// TIA Portal project "PLC - Mo hinh chiet rot" (V15)

(* hardware
DEVICE "S7-1200 station_1"  S7-1200 Station
   slot 0: "Rack_0"  S7-1200 Rack  Rack  V1.0
   slot 1: "PLC_1"  CPU 1212C AC/DC/Rly  6ES7 212-1BE40-0XB0  V4.2
   slot 2: "DQ 8xRelay_1"  SM 1222 DQ8 x relay  6ES7 222-1HF32-0XB0  V2.0
*)

// ===== PLC "PLC_1"  CPU 1212C AC/DC/Rly =====

VAR_GLOBAL   // PLC tag table "Default tag table"
   "CB1" AT %I0.0 : Bool;
   "CB2" AT %I0.1 : Bool;
   "CB3" AT %I0.2 : Bool;
   "CB4" AT %I0.3 : Bool;
   "Start" AT %I0.4 : Bool;
   "Stop" AT %I0.5 : Bool;
   "Reset" AT %I0.6 : Bool;
   "Emc" AT %I0.7 : Bool;
   "Van1" AT %Q0.0 : Bool;
   "Van2" AT %Q0.1 : Bool;
   "Van3" AT %Q0.2 : Bool;
   "Van4" AT %Q0.3 : Bool;
   "Van5" AT %Q0.4 : Bool;
   "Van6" AT %Q0.5 : Bool;
   "Step-M-MXoay" AT %Q1.0 : Bool;
   "Step-U-Dnhan" AT %Q1.7 : Bool;
   "DC1-M-BT1" AT %Q1.3 : Bool;
   "DC2-M-BT2" AT %Q1.4 : Bool;
   "DC3-M-CNap" AT %Q1.5 : Bool;
   "DC4-M-Bom" AT %Q1.6 : Bool;
   "DC5-U-BT3" AT %Q1.1 : Bool;
   "M-Start" AT %M0.0 : Bool;
   "M-Start3s" AT %M1.0 : Bool;
   "M-Bom" AT %M2.0 : Bool;
   "M-MX chay dien" AT %M1.1 : Bool;
   "M-MX chay" AT %M2.1 : Bool;
   "Tag_1" AT %M4.1 : Bool;
   "Tag_3" AT %M4.2 : Bool;
   "Tag_4" AT %MW10 : Int;
   "Tag_5" AT %M4.5 : Bool;
   "Tag_6" AT %M0.1 : Bool;
   "Tag_7" AT %M0.2 : Bool;
   "Tag_8" AT %M0.3 : Bool;
   "Tag_9" AT %M0.5 : Bool;
   "Tag_2" AT %M6.0 : Bool;
   "Tag_10" AT %M0.4 : Bool;
   "Tag_11" AT %M9.0 : Bool;
END_VAR

// folder: System blocks/Program resources

DATA_BLOCK "t1"   // DB1
{ S7_Optimized_Access := 'TRUE' }
AUTHOR : Simatic
FAMILY : IEC
NAME : IEC_TMR
VERSION : 1.0
// stored: InstanceOfName IEC_TIMER
"IEC_TIMER"
BEGIN
END_DATA_BLOCK

DATA_BLOCK "t2"   // DB2
{ S7_Optimized_Access := 'TRUE' }
AUTHOR : Simatic
FAMILY : IEC
NAME : IEC_TMR
VERSION : 1.0
// stored: InstanceOfName IEC_TIMER
"IEC_TIMER"
BEGIN
END_DATA_BLOCK

DATA_BLOCK "T0"   // DB3
{ S7_Optimized_Access := 'TRUE' }
AUTHOR : Simatic
FAMILY : IEC
NAME : IEC_TMR
VERSION : 1.0
// stored: InstanceOfName IEC_TIMER
"IEC_TIMER"
BEGIN
END_DATA_BLOCK

DATA_BLOCK "t3"   // DB4
{ S7_Optimized_Access := 'TRUE' }
AUTHOR : Simatic
FAMILY : IEC
NAME : IEC_TMR
VERSION : 1.0
// stored: InstanceOfName IEC_TIMER
"IEC_TIMER"
BEGIN
END_DATA_BLOCK

DATA_BLOCK "t9"   // DB5
{ S7_Optimized_Access := 'TRUE' }
AUTHOR : Simatic
FAMILY : IEC
NAME : IEC_TMR
VERSION : 1.0
// stored: InstanceOfName IEC_TIMER
"IEC_TIMER"
BEGIN
END_DATA_BLOCK

DATA_BLOCK "t5"   // DB6
{ S7_Optimized_Access := 'TRUE' }
AUTHOR : Simatic
FAMILY : IEC
NAME : IEC_TMR
VERSION : 1.0
// stored: InstanceOfName IEC_TIMER
"IEC_TIMER"
BEGIN
END_DATA_BLOCK

DATA_BLOCK "t6"   // DB7
{ S7_Optimized_Access := 'TRUE' }
AUTHOR : Simatic
FAMILY : IEC
NAME : IEC_TMR
VERSION : 1.0
// stored: InstanceOfName IEC_TIMER
"IEC_TIMER"
BEGIN
END_DATA_BLOCK

DATA_BLOCK "t7"   // DB8
{ S7_Optimized_Access := 'TRUE' }
AUTHOR : Simatic
FAMILY : IEC
NAME : IEC_TMR
VERSION : 1.0
// stored: InstanceOfName IEC_TIMER
"IEC_TIMER"
BEGIN
END_DATA_BLOCK

DATA_BLOCK "t8"   // DB9
{ S7_Optimized_Access := 'TRUE' }
AUTHOR : Simatic
FAMILY : IEC
NAME : IEC_TMR
VERSION : 1.0
// stored: InstanceOfName IEC_TIMER
"IEC_TIMER"
BEGIN
END_DATA_BLOCK

DATA_BLOCK "t10"   // DB10
{ S7_Optimized_Access := 'TRUE' }
AUTHOR : Simatic
FAMILY : IEC
NAME : IEC_TMR
VERSION : 1.0
// stored: InstanceOfName IEC_TIMER
"IEC_TIMER"
BEGIN
END_DATA_BLOCK

DATA_BLOCK "dem"   // DB11
{ S7_Optimized_Access := 'TRUE' }
AUTHOR : Simatic
FAMILY : IEC
NAME : CNTR
VERSION : 1.0
// stored: InstanceOfName IEC_COUNTER
"IEC_COUNTER"
BEGIN
END_DATA_BLOCK

DATA_BLOCK "t11"   // DB12
{ S7_Optimized_Access := 'TRUE' }
AUTHOR : Simatic
FAMILY : IEC
NAME : IEC_TMR
VERSION : 1.0
// stored: InstanceOfName IEC_TIMER
"IEC_TIMER"
BEGIN
END_DATA_BLOCK

DATA_BLOCK "t24"   // DB13
{ S7_Optimized_Access := 'TRUE' }
AUTHOR : Simatic
FAMILY : IEC
NAME : IEC_TMR
VERSION : 1.0
// stored: InstanceOfName IEC_TIMER
"IEC_TIMER"
BEGIN
END_DATA_BLOCK

DATA_BLOCK "t12"   // DB14
{ S7_Optimized_Access := 'TRUE' }
AUTHOR : Simatic
FAMILY : IEC
NAME : IEC_TMR
VERSION : 1.0
// stored: InstanceOfName IEC_TIMER
"IEC_TIMER"
BEGIN
END_DATA_BLOCK

DATA_BLOCK "t25"   // DB15
{ S7_Optimized_Access := 'TRUE' }
AUTHOR : Simatic
FAMILY : IEC
NAME : IEC_TMR
VERSION : 1.0
// stored: InstanceOfName IEC_TIMER
"IEC_TIMER"
BEGIN
END_DATA_BLOCK

DATA_BLOCK "t13"   // DB16
{ S7_Optimized_Access := 'TRUE' }
AUTHOR : Simatic
FAMILY : IEC
NAME : IEC_TMR
VERSION : 1.0
// stored: InstanceOfName IEC_TIMER
"IEC_TIMER"
BEGIN
END_DATA_BLOCK

DATA_BLOCK "t16"   // DB17
{ S7_Optimized_Access := 'TRUE' }
AUTHOR : Simatic
FAMILY : IEC
NAME : IEC_TMR
VERSION : 1.0
// stored: InstanceOfName IEC_TIMER
"IEC_TIMER"
BEGIN
END_DATA_BLOCK

DATA_BLOCK "t23"   // DB18
{ S7_Optimized_Access := 'TRUE' }
AUTHOR : Simatic
FAMILY : IEC
NAME : IEC_TMR
VERSION : 1.0
// stored: InstanceOfName IEC_TIMER
"IEC_TIMER"
BEGIN
END_DATA_BLOCK

DATA_BLOCK "t20"   // DB19
{ S7_Optimized_Access := 'TRUE' }
AUTHOR : Simatic
FAMILY : IEC
NAME : IEC_TMR
VERSION : 1.0
// stored: InstanceOfName IEC_TIMER
"IEC_TIMER"
BEGIN
END_DATA_BLOCK

DATA_BLOCK "t26"   // DB20
{ S7_Optimized_Access := 'TRUE' }
AUTHOR : Simatic
FAMILY : IEC
NAME : IEC_TMR
VERSION : 1.0
// stored: InstanceOfName IEC_TIMER
"IEC_TIMER"
BEGIN
END_DATA_BLOCK

DATA_BLOCK "t27"   // DB21
{ S7_Optimized_Access := 'TRUE' }
AUTHOR : Simatic
FAMILY : IEC
NAME : IEC_TMR
VERSION : 1.0
// stored: InstanceOfName IEC_TIMER
"IEC_TIMER"
BEGIN
END_DATA_BLOCK

// folder: (top level)

ORGANIZATION_BLOCK "Main"   // OB1, LAD, ProgramCycle
TITLE = "Main Program Sweep (Cycle)"
{ S7_Optimized_Access := 'TRUE' }
VERSION : 0.1
   VAR_INPUT
      Initial_Call : Bool;   // Initial call of this OB
      Remanence : Bool;   // =True, if remanent data are available
   END_VAR
   VAR_TEMP   // added for the SCL form of the ladder/FBD networks
      _w1 : Bool;
   END_VAR
BEGIN

REGION Network 1: start vs stop
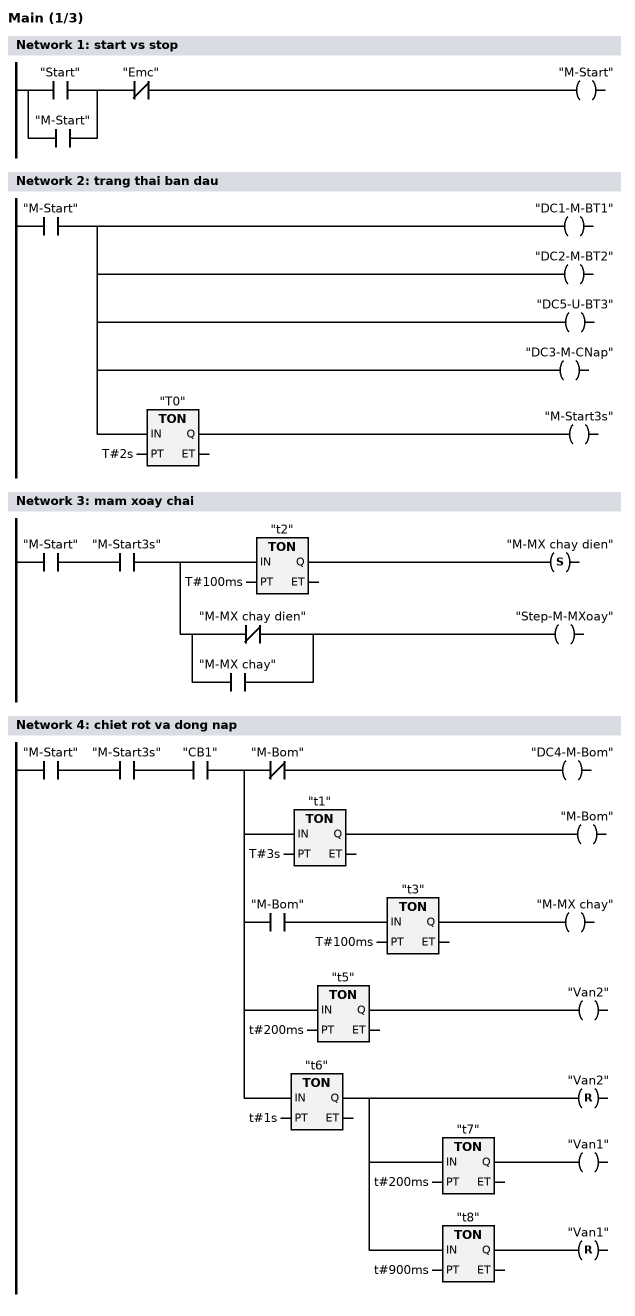
   RUNG wire#powerrail
      Contact( "Start" )
      wire#w1
      I_Contact( "Emc" )
      Coil( "M-Start" )
   END_RUNG
   RUNG wire#powerrail
      Contact( "M-Start" )
   END_RUNG wire#w1
   // the same network as SCL:
   "M-Start" := ("Start" OR "M-Start") AND NOT "Emc";
END_REGION

REGION Network 2: trang thai ban dau
   "DC1-M-BT1" := "M-Start";
   "DC2-M-BT2" := "M-Start";
   "DC5-U-BT3" := "M-Start";
   "DC3-M-CNap" := "M-Start";
   "T0".TON(IN := "M-Start", PT := T#2s);
   "M-Start3s" := "T0".Q;
END_REGION

REGION Network 3: mam xoay chai
   #_w1 := "M-Start" AND "M-Start3s";
   "t2".TON(IN := #_w1, PT := T#100ms);
   IF "t2".Q THEN "M-MX chay dien" := TRUE; END_IF;
   "Step-M-MXoay" := #_w1 AND (NOT "M-MX chay dien" OR "M-MX chay");
END_REGION

REGION Network 4: chiet rot va dong nap
   #_w1 := "M-Start" AND "M-Start3s" AND "CB1";
   "DC4-M-Bom" := #_w1 AND NOT "M-Bom";
   "t1".TON(IN := #_w1, PT := T#3s);
   "M-Bom" := "t1".Q;
   "t3".TON(IN := #_w1 AND "M-Bom", PT := T#100ms);
   "M-MX chay" := "t3".Q;
   "t5".TON(IN := #_w1, PT := t#200ms);
   "Van2" := "t5".Q;
   "t6".TON(IN := #_w1, PT := t#1s);
   IF "t6".Q THEN "Van2" := FALSE; END_IF;
   "t7".TON(IN := "t6".Q, PT := t#200ms);
   "Van1" := "t7".Q;
   "t8".TON(IN := "t6".Q, PT := t#900ms);
   IF "t8".Q THEN "Van1" := FALSE; END_IF;
END_REGION

REGION Network 5
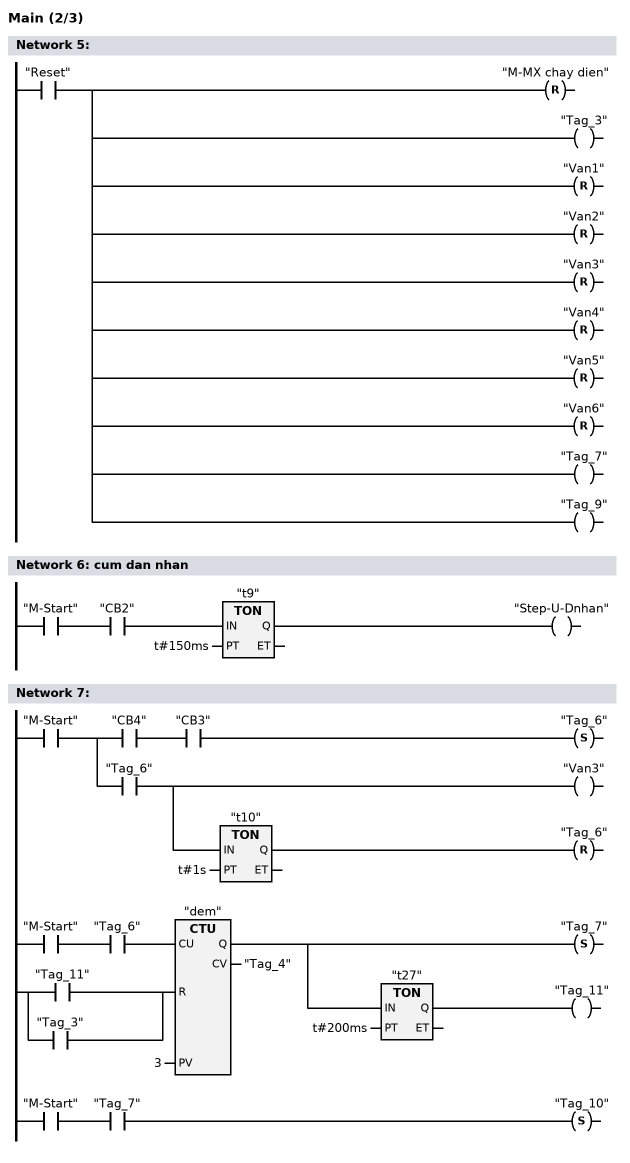
   RUNG wire#powerrail
      Contact( "Reset" )
      wire#w1
      R_Coil( "M-MX chay dien" )
   END_RUNG
   RUNG wire#w1
      Coil( "Tag_3" )
   END_RUNG
   RUNG wire#w1
      R_Coil( "Van1" )
   END_RUNG
   RUNG wire#w1
      R_Coil( "Van2" )
   END_RUNG
   RUNG wire#w1
      R_Coil( "Van3" )
   END_RUNG
   RUNG wire#w1
      R_Coil( "Van4" )
   END_RUNG
   RUNG wire#w1
      R_Coil( "Van5" )
   END_RUNG
   RUNG wire#w1
      R_Coil( "Van6" )
   END_RUNG
   RUNG wire#w1
      Coil( "Tag_7" )
   END_RUNG
   RUNG wire#w1
      Coil( "Tag_9" )
   END_RUNG
   // the same network as SCL:
   IF "Reset" THEN "M-MX chay dien" := FALSE; END_IF;
   "Tag_3" := "Reset";
   IF "Reset" THEN
       "Van1" := FALSE;
       "Van2" := FALSE;
       "Van3" := FALSE;
       "Van4" := FALSE;
       "Van5" := FALSE;
       "Van6" := FALSE;
   END_IF;
   "Tag_7" := "Reset";
   "Tag_9" := "Reset";
END_REGION

REGION Network 6: cum dan nhan
   "t9".TON(IN := "M-Start" AND "CB2", PT := t#150ms);
   "Step-U-Dnhan" := "t9".Q;
END_REGION

REGION Network 7
   IF "M-Start" AND "CB4" AND "CB3" THEN "Tag_6" := TRUE; END_IF;
   "Van3" := "M-Start" AND "Tag_6";
   "t10".TON(IN := "Van3", PT := t#1s);
   IF "t10".Q THEN "Tag_6" := FALSE; END_IF;
   "dem".CTU(CU := "M-Start" AND "Tag_6", R := "Tag_11" OR "Tag_3", PV := 3, CV => "Tag_4");
   IF "dem".Q THEN "Tag_7" := TRUE; END_IF;
   "t27".TON(IN := "dem".Q, PT := t#200ms);
   "Tag_11" := "t27".Q;
   IF "M-Start" AND "Tag_7" THEN "Tag_10" := TRUE; END_IF;
END_REGION

REGION Network 8: 6 chai
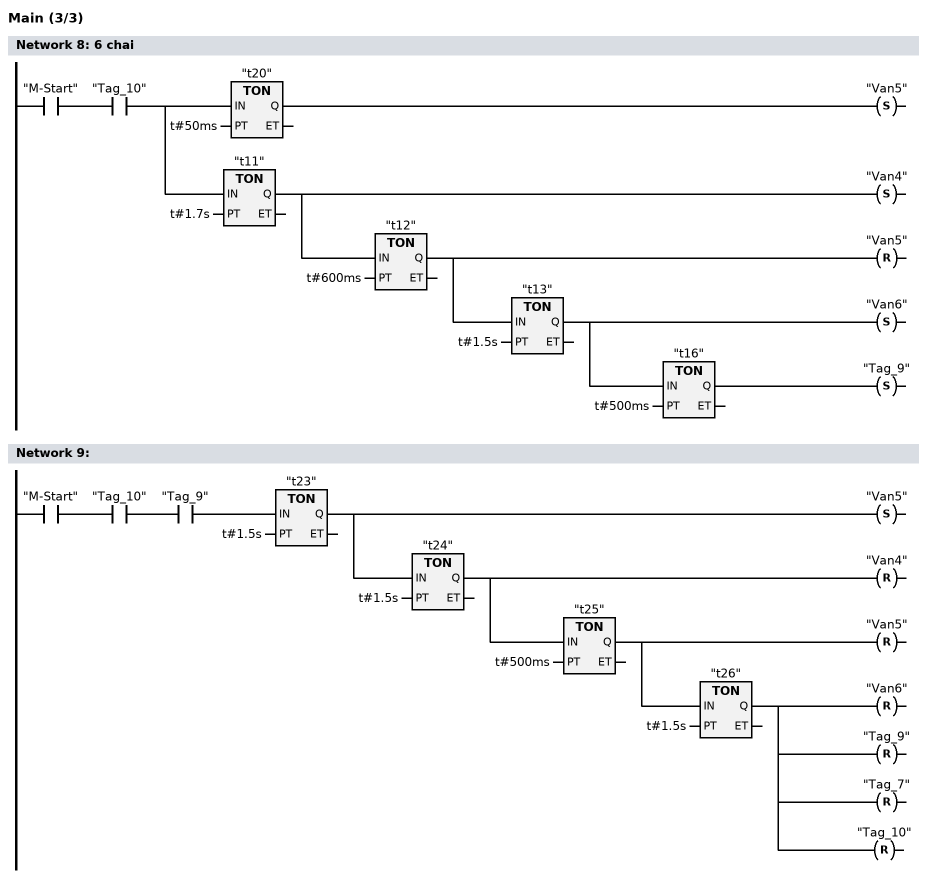
   #_w1 := "M-Start" AND "Tag_10";
   "t20".TON(IN := #_w1, PT := t#50ms);
   IF "t20".Q THEN "Van5" := TRUE; END_IF;
   "t11".TON(IN := #_w1, PT := t#1.7s);
   IF "t11".Q THEN "Van4" := TRUE; END_IF;
   "t12".TON(IN := "t11".Q, PT := t#600ms);
   IF "t12".Q THEN "Van5" := FALSE; END_IF;
   "t13".TON(IN := "t12".Q, PT := t#1.5s);
   IF "t13".Q THEN "Van6" := TRUE; END_IF;
   "t16".TON(IN := "t13".Q, PT := t#500ms);
   IF "t16".Q THEN "Tag_9" := TRUE; END_IF;
END_REGION

REGION Network 9
   "t23".TON(IN := "M-Start" AND "Tag_10" AND "Tag_9", PT := t#1.5s);
   IF "t23".Q THEN "Van5" := TRUE; END_IF;
   "t24".TON(IN := "t23".Q, PT := t#1.5s);
   IF "t24".Q THEN "Van4" := FALSE; END_IF;
   "t25".TON(IN := "t24".Q, PT := t#500ms);
   IF "t25".Q THEN "Van5" := FALSE; END_IF;
   "t26".TON(IN := "t25".Q, PT := t#1.5s);
   IF "t26".Q THEN
       "Van6" := FALSE;
       "Tag_9" := FALSE;
       "Tag_7" := FALSE;
       "Tag_10" := FALSE;
   END_IF;
END_REGION
END_ORGANIZATION_BLOCK